{attribute addProperty BoxType "EL3632-0000-0016"}
{attribute addProperty Id "Ch1_ValueAT %I*INT162"}
{attribute addProperty CRC "935361667"}
{attribute addProperty SizeInBites "16"}
{attribute addProperty SizeInBytes "2"}
TYPE Ch1_Sample_37C07C83 :
STRUCT
	{attribute addProperty Name "Ch1_Value"}
	Ch1_Value AT %I* : INT;
END_STRUCT
END_TYPE

(* stored: Version 1.2.0.0, ProductVersion 3.1.4024.9
   DUT Ch1_Sample_37C07C83: Id {2df0c0af-c2da-4b64-a644-78fcde5ff27f} *)
